Universal Robots PolyScope program: watering.urp

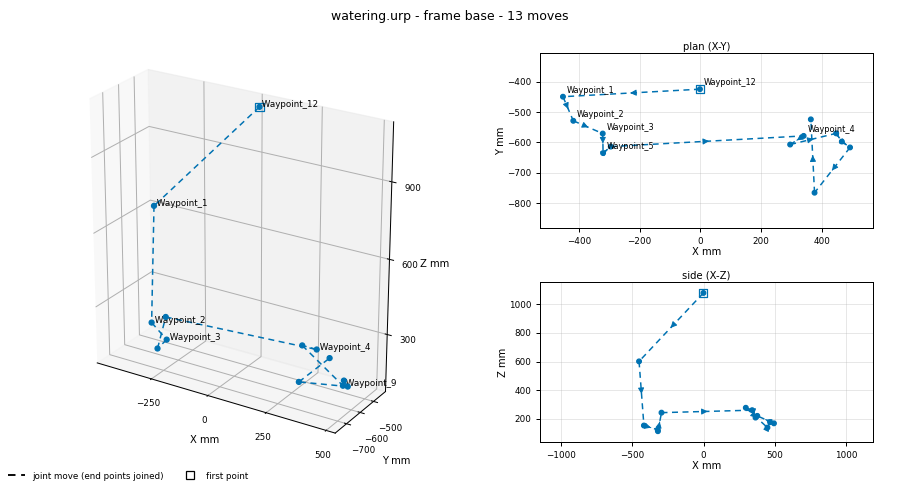
[picture p0: tool path of watering.urp in frame base, 13 of 13 moves have a stored position in this frame; points joined in program order, loops and branches not executed]
Program watering (installation=default directory=/programs/yutongxie createdIn=5.12.6.1102099 lastSavedIn=5.12.6.1102099 robotSerialNumber=20215500597)
Calibrated DH parameters: a=[0.000193, -0.066673, -0.391568, -0.000012, 0.00005, 0]; d=[0.162643, -472.05677, 465.132521, 7.058239, 0.099746, 0.099582]; alpha=[1.571116, 0.00089, 0.003862, 1.569269, -1.569248, 0]; deltaTheta=[0, -1.413394, 7.628392, 0.068187, 0, -0.000001]
Robot Program (runOnlyOnce=true)
  MoveJ speed 60 deg/s, acceleration 80 deg/s^2 (useActiveTCP=true) feature=Base
    Waypoint Waypoint_12: TCP in base x=-1.516 y=-424.817 z=1080.554 mm, rx=-0.0044 ry=-2.2185 rz=2.2204 rad; joints [0.001, -90.002, 0.002, -90, 0.001, 0.001] deg; TCP offset x=0 y=0 z=191.5 mm, rx=0 ry=0 rz=0 rad
    Waypoint Waypoint_1: TCP in base x=-452.58 y=-449.629 z=600.904 mm, rx=1.1637 ry=1.2668 rz=-1.1886 rad; joints [3.039, -92.191, 90.11, -89.817, -0.566, 0.03] deg
    Waypoint Waypoint_2: TCP in base x=-418.553 y=-528.931 z=151.395 mm, rx=1.5718 ry=0.1293 rz=0.1857 rad; joints [12.622, -56.769, 99.435, -40.974, 1.238, 0.39] deg
    URCap Gripper Activate (Robotiq_Grippers, Robotiq Inc.) dataModel(ResetAndActivateKey=false)
    URCap Gripper (Robotiq_Grippers, Robotiq Inc.) dataModel(position=1.1764705882352942, force=100.0, speed=100.0, positionInDouble=1.1764705882352942, forceInDouble=100.0, speedInDouble=100.0, slaveIds=[9], blocking=true)
    Waypoint Waypoint_3: TCP in base x=-321.664 y=-570.955 z=121.656 mm, rx=1.5454 ry=-0.0127 rz=-0.0059 rad; joints [22.929, -64.133, 121.715, -61.448, 23.812, 3.805] deg
    Waypoint Waypoint_5: TCP in base x=-320.473 y=-635.272 z=111.605 mm, rx=1.5506 ry=-0.0192 rz=0.0014 rad; joints [30.736, -58.94, 113.884, -57.357, 31.559, 2.834] deg
    URCap Gripper (Robotiq_Grippers, Robotiq Inc.) dataModel(position=100.0, force=100.0, speed=0.0, positionInDouble=100.0, forceInDouble=100.0, speedInDouble=0.0, slaveIds=[9], blocking=true)
    Waypoint Waypoint_6: TCP in base x=-295.301 y=-613.867 z=241.631 mm, rx=1.5646 ry=0.016 rz=-0.0806 rad; joints [30.598, -77.139, 114.378, -38.203, 33.053, -2.674] deg
    Waypoint Waypoint_4: TCP in base x=339.944 y=-578.671 z=258.938 mm, rx=1.3941 ry=0.8462 rz=0.793 rad; joints [83.724, -76.893, 110.447, -33.513, 23.366, -2.072] deg
    Waypoint Waypoint_7: TCP in base x=295.565 y=-607.115 z=275.813 mm, rx=1.9176 ry=-0.5578 rz=1.835 rad; joints [79.622, -77.376, 106.632, -24.67, 23.847, 84.19] deg
    Waypoint Waypoint_9: TCP in base x=447.16 y=-570.259 z=136.967 mm, rx=2.1076 ry=-0.3588 rz=2.0148 rad; joints [94.385, -58.374, 102.732, -37.57, 22.783, 84.936] deg
    Waypoint water_collect: TCP in base x=465.696 y=-597.188 z=174.832 mm, rx=-2.0351 ry=0.9984 rz=-2.1707 rad; joints [98.38, -61.94, 101.636, -35.575, 34.551, 112.9] deg
    Wait Sleep waitTime=7
    Waypoint Waypoint_8: TCP in base x=492.734 y=-616.705 z=166.731 mm, rx=-2.0351 ry=0.9985 rz=-2.1705 rad; joints [101.011, -58.124, 96.669, -34.669, 37.167, 113.218] deg
    Waypoint Waypoint_10: TCP in base x=375.858 y=-765.72 z=219.063 mm, rx=-0.6277 ry=1.4901 rz=-1.3781 rad; joints [88.511, -50.027, 81.848, -47.642, 25.923, 212.168] deg
    Wait Sleep waitTime=7
    Waypoint Waypoint_11: TCP in base x=363.654 y=-524.221 z=206.978 mm, rx=-2.1294 ry=-0.3551 rz=-1.9842 rad; joints [85.734, -55.086, 83.179, -38.365, -22.833, 98.806] deg
